PROGRAM Test_AnalogInput
VAR
	fbLoadCell : FB_AnalogLoadCellInput; 
	rOutputNewtons : REAL; 
END_VAR

fbLoadCell(); 
rOutputNewtons := fbLoadCell.rCalibratedOutput;

END_PROGRAM

(* stored: Version 1.1.0.1, ProductVersion 3.1.4024.12
   POU Test_AnalogInput: Id {5a628192-256d-4a4c-abb8-e8dbd9f140a1}, SpecialFunc None *)
